// TIA Portal V17 export
// export: Created 2024-09-02T12:50:06.9482264Z, ExportSetting WithDefaults, DisplayName Totally Integrated Automation Portal, DisplayVersion V17, DisplayName TIA Portal Openness, DisplayVersion V17, DisplayName TIA Portal Version Control Interface, DisplayVersion V17, DisplayName STEP 7 Professional, DisplayVersion V17, DisplayName STEP 7 Safety, DisplayVersion V17, DisplayName WinCC Professional, DisplayVersion V17
FUNCTION "AnwFC1_FG01_Transport_OP70" : Void   // FC1281, LAD
TITLE = Transport
{ S7_Optimized_Access := 'TRUE' }
AUTHOR : VAF
FAMILY : SK
NAME : SK
VERSION : 0.1
// stored: AutoNumber false, IsIECCheckEnabled false, SetENOAutomatically false, UDAEnableTagReadback false
   VAR_TEMP
      Motion_Release : Bool;   // Motion permit
      Hand : Bool;
      Auto : Bool;
      t_ParityFault : Bool;
      t_ConfigFault : Bool;
      t_retval : Bool;
      "MM30/31_Home" : Bool;
      "MM30/31_Work" : Bool;
   END_VAR
BEGIN

REGION Network 1: Motion permit / Hand/ Auto
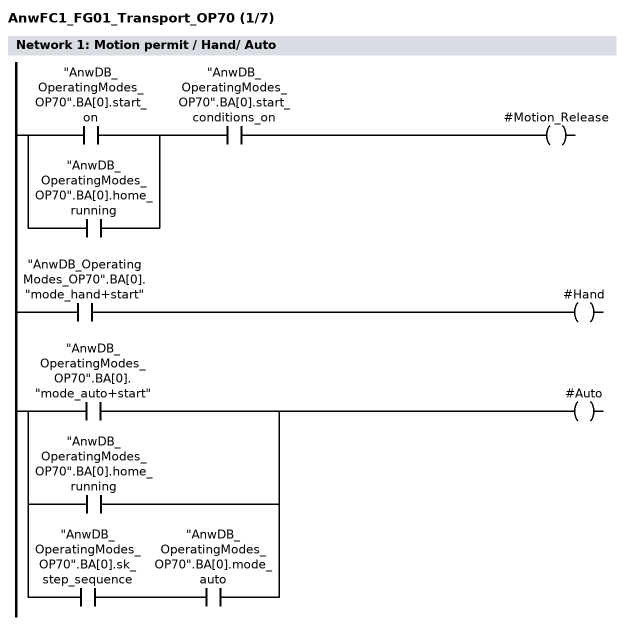
   RUNG wire#powerrail
      Contact( "AnwDB_OperatingModes_OP70".BA[0].start_on )
      wire#w1
      Contact( "AnwDB_OperatingModes_OP70".BA[0].start_conditions_on )
      Coil( #Motion_Release )
   END_RUNG
   RUNG wire#powerrail
      Contact( "AnwDB_OperatingModes_OP70".BA[0].home_running )
   END_RUNG wire#w1
   RUNG wire#powerrail
      Contact( "AnwDB_OperatingModes_OP70".BA[0]."mode_hand+start" )
      Coil( #Hand )
   END_RUNG
   RUNG wire#powerrail
      Contact( "AnwDB_OperatingModes_OP70".BA[0]."mode_auto+start" )
      wire#w2
      Coil( #Auto )
   END_RUNG
   RUNG wire#powerrail
      Contact( "AnwDB_OperatingModes_OP70".BA[0].home_running )
   END_RUNG wire#w2
   RUNG wire#powerrail
      Contact( "AnwDB_OperatingModes_OP70".BA[0].sk_step_sequence )
      Contact( "AnwDB_OperatingModes_OP70".BA[0].mode_auto )
   END_RUNG wire#w2
   // the same network as SCL:
   #Motion_Release := ("AnwDB_OperatingModes_OP70".BA[0].start_on OR "AnwDB_OperatingModes_OP70".BA[0].home_running) AND "AnwDB_OperatingModes_OP70".BA[0].start_conditions_on;
   #Hand := "AnwDB_OperatingModes_OP70".BA[0]."mode_hand+start";
   #Auto := "AnwDB_OperatingModes_OP70".BA[0]."mode_auto+start" OR "AnwDB_OperatingModes_OP70".BA[0].home_running OR ("AnwDB_OperatingModes_OP70".BA[0].sk_step_sequence AND "AnwDB_OperatingModes_OP70".BA[0].mode_auto);
END_REGION

REGION Network 2: Call of the step sequence
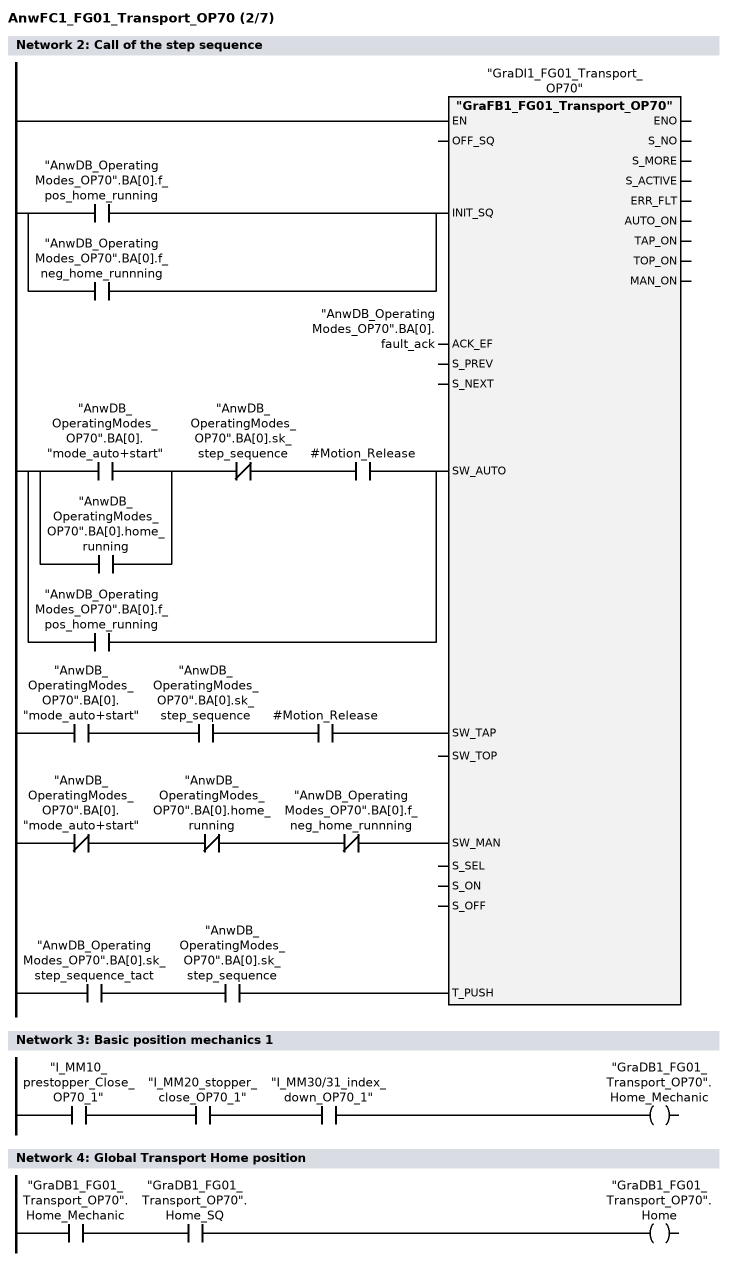
   RUNG wire#powerrail
      "GraDI1_FG01_Transport_OP70"(INIT_SQ := wire#w1, SW_AUTO := wire#w3, SW_TAP := wire#w4, SW_MAN := wire#w5, T_PUSH := wire#w6, OFF_SQ :=, ACK_EF := "AnwDB_OperatingModes_OP70".BA[0].fault_ack, S_PREV :=, S_NEXT :=, SW_TOP :=, S_SEL :=, S_ON :=, S_OFF :=, S_NO =>, S_MORE =>, S_ACTIVE =>, ERR_FLT =>, AUTO_ON =>, TAP_ON =>, TOP_ON =>, MAN_ON =>)
   END_RUNG
   RUNG wire#powerrail
      Contact( "AnwDB_OperatingModes_OP70".BA[0].f_pos_home_running )
   END_RUNG wire#w1
   RUNG wire#powerrail
      Contact( "AnwDB_OperatingModes_OP70".BA[0].f_neg_home_runnning )
   END_RUNG wire#w1
   RUNG wire#powerrail
      Contact( "AnwDB_OperatingModes_OP70".BA[0]."mode_auto+start" )
      wire#w2
      I_Contact( "AnwDB_OperatingModes_OP70".BA[0].sk_step_sequence )
      Contact( #Motion_Release )
   END_RUNG wire#w3
   RUNG wire#powerrail
      Contact( "AnwDB_OperatingModes_OP70".BA[0].home_running )
   END_RUNG wire#w2
   RUNG wire#powerrail
      Contact( "AnwDB_OperatingModes_OP70".BA[0].f_pos_home_running )
   END_RUNG wire#w3
   RUNG wire#powerrail
      Contact( "AnwDB_OperatingModes_OP70".BA[0]."mode_auto+start" )
      Contact( "AnwDB_OperatingModes_OP70".BA[0].sk_step_sequence )
      Contact( #Motion_Release )
   END_RUNG wire#w4
   RUNG wire#powerrail
      I_Contact( "AnwDB_OperatingModes_OP70".BA[0]."mode_auto+start" )
      I_Contact( "AnwDB_OperatingModes_OP70".BA[0].home_running )
      I_Contact( "AnwDB_OperatingModes_OP70".BA[0].f_neg_home_runnning )
   END_RUNG wire#w5
   RUNG wire#powerrail
      Contact( "AnwDB_OperatingModes_OP70".BA[0].sk_step_sequence_tact )
      Contact( "AnwDB_OperatingModes_OP70".BA[0].sk_step_sequence )
   END_RUNG wire#w6
   // the same network as SCL:
   "GraDI1_FG01_Transport_OP70"(INIT_SQ := "AnwDB_OperatingModes_OP70".BA[0].f_pos_home_running OR "AnwDB_OperatingModes_OP70".BA[0].f_neg_home_runnning,   // "GraFB1_FG01_Transport_OP70"
                           ACK_EF := "AnwDB_OperatingModes_OP70".BA[0].fault_ack,
                           SW_AUTO := (("AnwDB_OperatingModes_OP70".BA[0]."mode_auto+start" OR "AnwDB_OperatingModes_OP70".BA[0].home_running) AND NOT "AnwDB_OperatingModes_OP70".BA[0].sk_step_sequence AND #Motion_Release) OR "AnwDB_OperatingModes_OP70".BA[0].f_pos_home_running,
                           SW_TAP := "AnwDB_OperatingModes_OP70".BA[0]."mode_auto+start" AND "AnwDB_OperatingModes_OP70".BA[0].sk_step_sequence AND #Motion_Release,
                           SW_MAN := NOT "AnwDB_OperatingModes_OP70".BA[0]."mode_auto+start" AND NOT "AnwDB_OperatingModes_OP70".BA[0].home_running AND NOT "AnwDB_OperatingModes_OP70".BA[0].f_neg_home_runnning,
                           T_PUSH := "AnwDB_OperatingModes_OP70".BA[0].sk_step_sequence_tact AND "AnwDB_OperatingModes_OP70".BA[0].sk_step_sequence);
END_REGION

REGION Network 3: Basic position mechanics 1
   RUNG wire#powerrail
      Contact( "I_MM10_prestopper_Close_OP70_1" )
      Contact( "I_MM20_stopper_close_OP70_1" )
      Contact( "I_MM30/31_index_down_OP70_1" )
      Coil( "GraDB1_FG01_Transport_OP70".Home_Mechanic )
   END_RUNG
   // the same network as SCL:
   "GraDB1_FG01_Transport_OP70".Home_Mechanic := "I_MM10_prestopper_Close_OP70_1" AND "I_MM20_stopper_close_OP70_1" AND "I_MM30/31_index_down_OP70_1";
END_REGION

REGION Network 4: Global Transport Home position
   RUNG wire#powerrail
      Contact( "GraDB1_FG01_Transport_OP70".Home_Mechanic )
      Contact( "GraDB1_FG01_Transport_OP70".Home_SQ )
      Coil( "GraDB1_FG01_Transport_OP70".Home )
   END_RUNG
   // the same network as SCL:
   "GraDB1_FG01_Transport_OP70".Home := "GraDB1_FG01_Transport_OP70".Home_Mechanic AND "GraDB1_FG01_Transport_OP70".Home_SQ;
END_REGION

REGION Network 5: Finished message OK
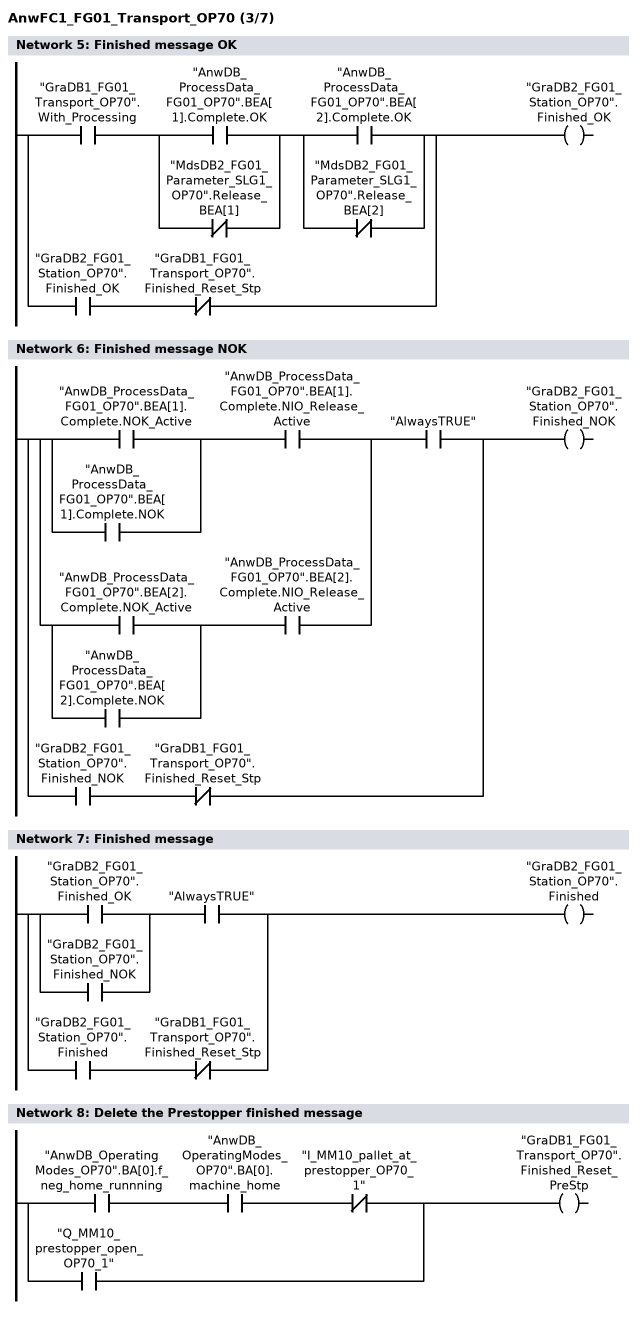
   RUNG wire#powerrail
      Contact( "GraDB1_FG01_Transport_OP70".With_Processing )
      wire#w1
      Contact( "AnwDB_ProcessData_FG01_OP70".BEA[1].Complete.OK )
      wire#w2
      Contact( "AnwDB_ProcessData_FG01_OP70".BEA[2].Complete.OK )
      wire#w3
      Coil( "GraDB2_FG01_Station_OP70".Finished_OK )
   END_RUNG
   RUNG wire#w1
      I_Contact( "MdsDB2_FG01_Parameter_SLG1_OP70".Release_BEA[1] )
   END_RUNG wire#w2
   RUNG wire#w2
      I_Contact( "MdsDB2_FG01_Parameter_SLG1_OP70".Release_BEA[2] )
   END_RUNG wire#w3
   RUNG wire#powerrail
      Contact( "GraDB2_FG01_Station_OP70".Finished_OK )
      I_Contact( "GraDB1_FG01_Transport_OP70".Finished_Reset_Stp )
   END_RUNG wire#w3
   // the same network as SCL:
   "GraDB2_FG01_Station_OP70".Finished_OK := ("GraDB1_FG01_Transport_OP70".With_Processing AND ("AnwDB_ProcessData_FG01_OP70".BEA[1].Complete.OK OR NOT "MdsDB2_FG01_Parameter_SLG1_OP70".Release_BEA[1]) AND ("AnwDB_ProcessData_FG01_OP70".BEA[2].Complete.OK OR NOT "MdsDB2_FG01_Parameter_SLG1_OP70".Release_BEA[2])) OR ("GraDB2_FG01_Station_OP70".Finished_OK AND NOT "GraDB1_FG01_Transport_OP70".Finished_Reset_Stp);
END_REGION

REGION Network 6: Finished message NOK
   RUNG wire#powerrail
      Contact( "AnwDB_ProcessData_FG01_OP70".BEA[1].Complete.NOK_Active )
      wire#w1
      Contact( "AnwDB_ProcessData_FG01_OP70".BEA[1].Complete.NIO_Release_Active )
      wire#w2
      Contact( "AlwaysTRUE" )
      wire#w4
      Coil( "GraDB2_FG01_Station_OP70".Finished_NOK )
   END_RUNG
   RUNG wire#powerrail
      Contact( "AnwDB_ProcessData_FG01_OP70".BEA[1].Complete.NOK )
   END_RUNG wire#w1
   RUNG wire#powerrail
      Contact( "AnwDB_ProcessData_FG01_OP70".BEA[2].Complete.NOK_Active )
      wire#w3
      Contact( "AnwDB_ProcessData_FG01_OP70".BEA[2].Complete.NIO_Release_Active )
   END_RUNG wire#w2
   RUNG wire#powerrail
      Contact( "AnwDB_ProcessData_FG01_OP70".BEA[2].Complete.NOK )
   END_RUNG wire#w3
   RUNG wire#powerrail
      Contact( "GraDB2_FG01_Station_OP70".Finished_NOK )
      I_Contact( "GraDB1_FG01_Transport_OP70".Finished_Reset_Stp )
   END_RUNG wire#w4
   // the same network as SCL:
   "GraDB2_FG01_Station_OP70".Finished_NOK := (((("AnwDB_ProcessData_FG01_OP70".BEA[1].Complete.NOK_Active OR "AnwDB_ProcessData_FG01_OP70".BEA[1].Complete.NOK) AND "AnwDB_ProcessData_FG01_OP70".BEA[1].Complete.NIO_Release_Active) OR (("AnwDB_ProcessData_FG01_OP70".BEA[2].Complete.NOK_Active OR "AnwDB_ProcessData_FG01_OP70".BEA[2].Complete.NOK) AND "AnwDB_ProcessData_FG01_OP70".BEA[2].Complete.NIO_Release_Active)) AND "AlwaysTRUE") OR ("GraDB2_FG01_Station_OP70".Finished_NOK AND NOT "GraDB1_FG01_Transport_OP70".Finished_Reset_Stp);
END_REGION

REGION Network 7: Finished message
   RUNG wire#powerrail
      Contact( "GraDB2_FG01_Station_OP70".Finished_OK )
      wire#w1
      Contact( "AlwaysTRUE" )
      wire#w2
      Coil( "GraDB2_FG01_Station_OP70".Finished )
   END_RUNG
   RUNG wire#powerrail
      Contact( "GraDB2_FG01_Station_OP70".Finished_NOK )
   END_RUNG wire#w1
   RUNG wire#powerrail
      Contact( "GraDB2_FG01_Station_OP70".Finished )
      I_Contact( "GraDB1_FG01_Transport_OP70".Finished_Reset_Stp )
   END_RUNG wire#w2
   // the same network as SCL:
   "GraDB2_FG01_Station_OP70".Finished := (("GraDB2_FG01_Station_OP70".Finished_OK OR "GraDB2_FG01_Station_OP70".Finished_NOK) AND "AlwaysTRUE") OR ("GraDB2_FG01_Station_OP70".Finished AND NOT "GraDB1_FG01_Transport_OP70".Finished_Reset_Stp);
END_REGION

REGION Network 8: Delete the Prestopper finished message
   RUNG wire#powerrail
      Contact( "AnwDB_OperatingModes_OP70".BA[0].f_neg_home_runnning )
      Contact( "AnwDB_OperatingModes_OP70".BA[0].machine_home )
      I_Contact( "I_MM10_pallet_at_prestopper_OP70_1" )
      wire#w1
      Coil( "GraDB1_FG01_Transport_OP70".Finished_Reset_PreStp )
   END_RUNG
   RUNG wire#powerrail
      Contact( "Q_MM10_prestopper_open_OP70_1" )
   END_RUNG wire#w1
   // the same network as SCL:
   "GraDB1_FG01_Transport_OP70".Finished_Reset_PreStp := ("AnwDB_OperatingModes_OP70".BA[0].f_neg_home_runnning AND "AnwDB_OperatingModes_OP70".BA[0].machine_home AND NOT "I_MM10_pallet_at_prestopper_OP70_1") OR "Q_MM10_prestopper_open_OP70_1";
END_REGION

REGION Network 9: Delete the stopper finished message
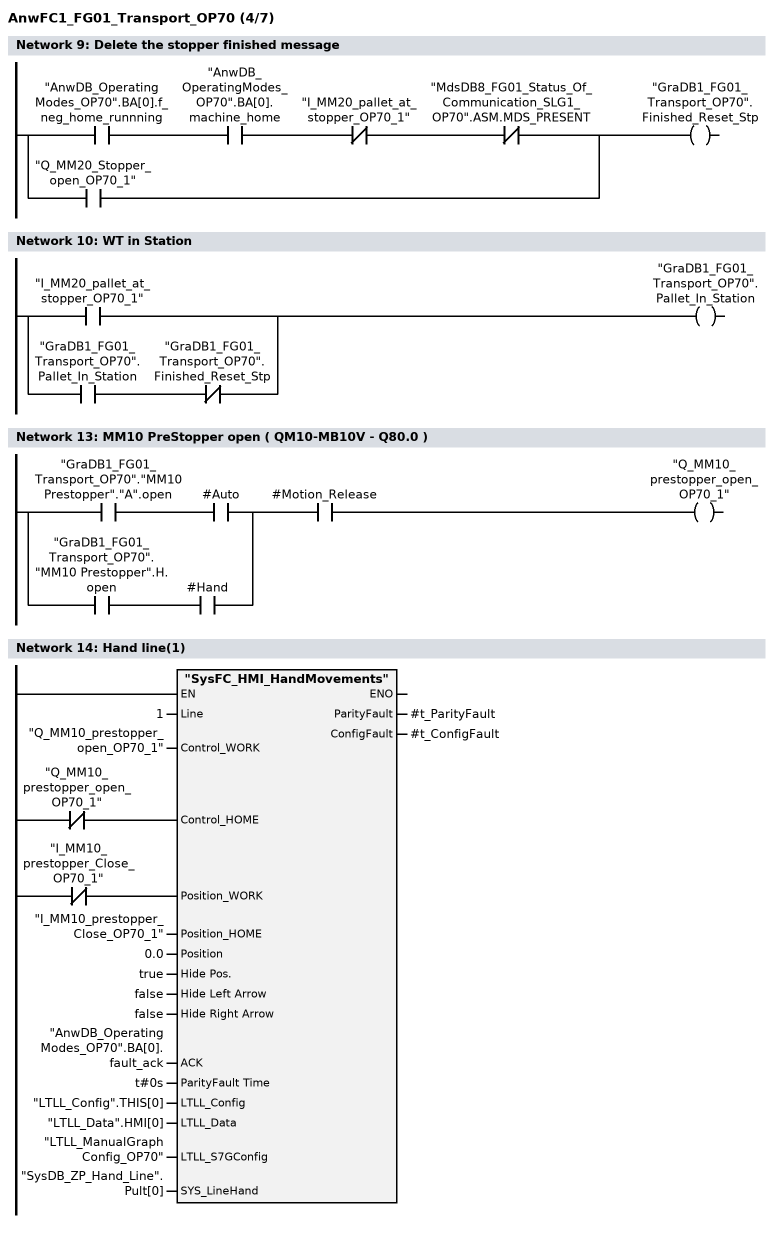
   RUNG wire#powerrail
      Contact( "AnwDB_OperatingModes_OP70".BA[0].f_neg_home_runnning )
      Contact( "AnwDB_OperatingModes_OP70".BA[0].machine_home )
      I_Contact( "I_MM20_pallet_at_stopper_OP70_1" )
      I_Contact( "MdsDB8_FG01_Status_Of_Communication_SLG1_OP70".ASM.MDS_PRESENT )
      wire#w1
      Coil( "GraDB1_FG01_Transport_OP70".Finished_Reset_Stp )
   END_RUNG
   RUNG wire#powerrail
      Contact( "Q_MM20_Stopper_open_OP70_1" )
   END_RUNG wire#w1
   // the same network as SCL:
   "GraDB1_FG01_Transport_OP70".Finished_Reset_Stp := ("AnwDB_OperatingModes_OP70".BA[0].f_neg_home_runnning AND "AnwDB_OperatingModes_OP70".BA[0].machine_home AND NOT "I_MM20_pallet_at_stopper_OP70_1" AND NOT "MdsDB8_FG01_Status_Of_Communication_SLG1_OP70".ASM.MDS_PRESENT) OR "Q_MM20_Stopper_open_OP70_1";
END_REGION

REGION Network 10: WT in Station
   RUNG wire#powerrail
      Contact( "I_MM20_pallet_at_stopper_OP70_1" )
      wire#w1
      Coil( "GraDB1_FG01_Transport_OP70".Pallet_In_Station )
   END_RUNG
   RUNG wire#powerrail
      Contact( "GraDB1_FG01_Transport_OP70".Pallet_In_Station )
      I_Contact( "GraDB1_FG01_Transport_OP70".Finished_Reset_Stp )
   END_RUNG wire#w1
   // the same network as SCL:
   "GraDB1_FG01_Transport_OP70".Pallet_In_Station := "I_MM20_pallet_at_stopper_OP70_1" OR ("GraDB1_FG01_Transport_OP70".Pallet_In_Station AND NOT "GraDB1_FG01_Transport_OP70".Finished_Reset_Stp);
END_REGION

REGION Network 11: ########### USER ###########
END_REGION

REGION Network 12: ########### SS_02_001_Setup ###########
END_REGION

REGION Network 13: MM10 PreStopper open ( QM10-MB10V - Q80.0 )
   RUNG wire#powerrail
      Contact( "GraDB1_FG01_Transport_OP70"."MM10 Prestopper"."A".open )
      Contact( #Auto )
      wire#w1
      Contact( #Motion_Release )
      Coil( "Q_MM10_prestopper_open_OP70_1" )
   END_RUNG
   RUNG wire#powerrail
      Contact( "GraDB1_FG01_Transport_OP70"."MM10 Prestopper".H.open )
      Contact( #Hand )
   END_RUNG wire#w1
   // the same network as SCL:
   "Q_MM10_prestopper_open_OP70_1" := (("GraDB1_FG01_Transport_OP70"."MM10 Prestopper"."A".open AND #Auto) OR ("GraDB1_FG01_Transport_OP70"."MM10 Prestopper".H.open AND #Hand)) AND #Motion_Release;
END_REGION

REGION Network 14: Hand line(1)
   RUNG wire#powerrail
      "SysFC_HMI_HandMovements"(Control_HOME := wire#w1, Position_WORK := wire#w2, Line := 1, Control_WORK := "Q_MM10_prestopper_open_OP70_1", Position_HOME := "I_MM10_prestopper_Close_OP70_1", Position := 0.0, "Hide Pos." := true, "Hide Left Arrow" := false, "Hide Right Arrow" := false, ACK := "AnwDB_OperatingModes_OP70".BA[0].fault_ack, "ParityFault Time" := t#0s, LTLL_Config := "LTLL_Config".THIS[0], LTLL_Data := "LTLL_Data".HMI[0], LTLL_S7GConfig := "LTLL_ManualGraphConfig_OP70", SYS_LineHand := "SysDB_ZP_Hand_Line".Pult[0], ParityFault => #t_ParityFault, ConfigFault => #t_ConfigFault)
   END_RUNG
   RUNG wire#powerrail
      I_Contact( "Q_MM10_prestopper_open_OP70_1" )
   END_RUNG wire#w1
   RUNG wire#powerrail
      I_Contact( "I_MM10_prestopper_Close_OP70_1" )
   END_RUNG wire#w2
   // the same network as SCL:
   "SysFC_HMI_HandMovements"(Line := 1,
                           Control_WORK := "Q_MM10_prestopper_open_OP70_1",
                           Control_HOME := NOT "Q_MM10_prestopper_open_OP70_1",
                           Position_WORK := NOT "I_MM10_prestopper_Close_OP70_1",
                           Position_HOME := "I_MM10_prestopper_Close_OP70_1",
                           Position := 0.0,
                           "Hide Pos." := true,
                           "Hide Left Arrow" := false,
                           "Hide Right Arrow" := false,
                           ACK := "AnwDB_OperatingModes_OP70".BA[0].fault_ack,
                           "ParityFault Time" := t#0s,
                           LTLL_Config := "LTLL_Config".THIS[0],
                           LTLL_Data := "LTLL_Data".HMI[0],
                           LTLL_S7GConfig := "LTLL_ManualGraphConfig_OP70",
                           SYS_LineHand := "SysDB_ZP_Hand_Line".Pult[0],
                           ParityFault => #t_ParityFault,
                           ConfigFault => #t_ConfigFault);
END_REGION

REGION Network 15: MM20 Stopper open ( QM20-MB20V - Q80.2 )
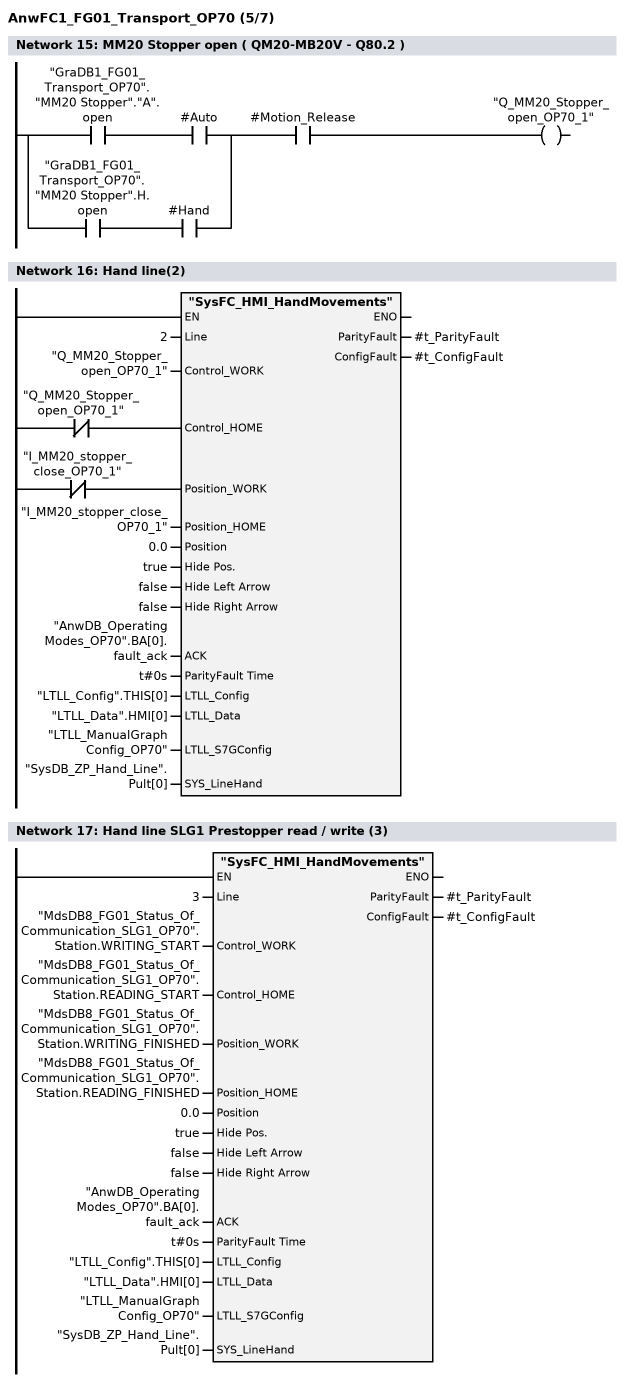
   RUNG wire#powerrail
      Contact( "GraDB1_FG01_Transport_OP70"."MM20 Stopper"."A".open )
      Contact( #Auto )
      wire#w1
      Contact( #Motion_Release )
      Coil( "Q_MM20_Stopper_open_OP70_1" )
   END_RUNG
   RUNG wire#powerrail
      Contact( "GraDB1_FG01_Transport_OP70"."MM20 Stopper".H.open )
      Contact( #Hand )
   END_RUNG wire#w1
   // the same network as SCL:
   "Q_MM20_Stopper_open_OP70_1" := (("GraDB1_FG01_Transport_OP70"."MM20 Stopper"."A".open AND #Auto) OR ("GraDB1_FG01_Transport_OP70"."MM20 Stopper".H.open AND #Hand)) AND #Motion_Release;
END_REGION

REGION Network 16: Hand line(2)
   RUNG wire#powerrail
      "SysFC_HMI_HandMovements"(Control_HOME := wire#w1, Position_WORK := wire#w2, Line := 2, Control_WORK := "Q_MM20_Stopper_open_OP70_1", Position_HOME := "I_MM20_stopper_close_OP70_1", Position := 0.0, "Hide Pos." := true, "Hide Left Arrow" := false, "Hide Right Arrow" := false, ACK := "AnwDB_OperatingModes_OP70".BA[0].fault_ack, "ParityFault Time" := t#0s, LTLL_Config := "LTLL_Config".THIS[0], LTLL_Data := "LTLL_Data".HMI[0], LTLL_S7GConfig := "LTLL_ManualGraphConfig_OP70", SYS_LineHand := "SysDB_ZP_Hand_Line".Pult[0], ParityFault => #t_ParityFault, ConfigFault => #t_ConfigFault)
   END_RUNG
   RUNG wire#powerrail
      I_Contact( "Q_MM20_Stopper_open_OP70_1" )
   END_RUNG wire#w1
   RUNG wire#powerrail
      I_Contact( "I_MM20_stopper_close_OP70_1" )
   END_RUNG wire#w2
   // the same network as SCL:
   "SysFC_HMI_HandMovements"(Line := 2,
                           Control_WORK := "Q_MM20_Stopper_open_OP70_1",
                           Control_HOME := NOT "Q_MM20_Stopper_open_OP70_1",
                           Position_WORK := NOT "I_MM20_stopper_close_OP70_1",
                           Position_HOME := "I_MM20_stopper_close_OP70_1",
                           Position := 0.0,
                           "Hide Pos." := true,
                           "Hide Left Arrow" := false,
                           "Hide Right Arrow" := false,
                           ACK := "AnwDB_OperatingModes_OP70".BA[0].fault_ack,
                           "ParityFault Time" := t#0s,
                           LTLL_Config := "LTLL_Config".THIS[0],
                           LTLL_Data := "LTLL_Data".HMI[0],
                           LTLL_S7GConfig := "LTLL_ManualGraphConfig_OP70",
                           SYS_LineHand := "SysDB_ZP_Hand_Line".Pult[0],
                           ParityFault => #t_ParityFault,
                           ConfigFault => #t_ConfigFault);
END_REGION

REGION Network 17: Hand line SLG1 Prestopper read / write (3)
   RUNG wire#powerrail
      "SysFC_HMI_HandMovements"(Line := 3, Control_WORK := "MdsDB8_FG01_Status_Of_Communication_SLG1_OP70".Station.WRITING_START, Control_HOME := "MdsDB8_FG01_Status_Of_Communication_SLG1_OP70".Station.READING_START, Position_WORK := "MdsDB8_FG01_Status_Of_Communication_SLG1_OP70".Station.WRITING_FINISHED, Position_HOME := "MdsDB8_FG01_Status_Of_Communication_SLG1_OP70".Station.READING_FINISHED, Position := 0.0, "Hide Pos." := true, "Hide Left Arrow" := false, "Hide Right Arrow" := false, ACK := "AnwDB_OperatingModes_OP70".BA[0].fault_ack, "ParityFault Time" := t#0s, LTLL_Config := "LTLL_Config".THIS[0], LTLL_Data := "LTLL_Data".HMI[0], LTLL_S7GConfig := "LTLL_ManualGraphConfig_OP70", SYS_LineHand := "SysDB_ZP_Hand_Line".Pult[0], ParityFault => #t_ParityFault, ConfigFault => #t_ConfigFault)
   END_RUNG
   // the same network as SCL:
   "SysFC_HMI_HandMovements"(Line := 3,
                           Control_WORK := "MdsDB8_FG01_Status_Of_Communication_SLG1_OP70".Station.WRITING_START,
                           Control_HOME := "MdsDB8_FG01_Status_Of_Communication_SLG1_OP70".Station.READING_START,
                           Position_WORK := "MdsDB8_FG01_Status_Of_Communication_SLG1_OP70".Station.WRITING_FINISHED,
                           Position_HOME := "MdsDB8_FG01_Status_Of_Communication_SLG1_OP70".Station.READING_FINISHED,
                           Position := 0.0,
                           "Hide Pos." := true,
                           "Hide Left Arrow" := false,
                           "Hide Right Arrow" := false,
                           ACK := "AnwDB_OperatingModes_OP70".BA[0].fault_ack,
                           "ParityFault Time" := t#0s,
                           LTLL_Config := "LTLL_Config".THIS[0],
                           LTLL_Data := "LTLL_Data".HMI[0],
                           LTLL_S7GConfig := "LTLL_ManualGraphConfig_OP70",
                           SYS_LineHand := "SysDB_ZP_Hand_Line".Pult[0],
                           ParityFault => #t_ParityFault,
                           ConfigFault => #t_ConfigFault);
END_REGION

REGION Network 18: MM30/31 Index unit up ( QM30-MB30V - Q81.0 )
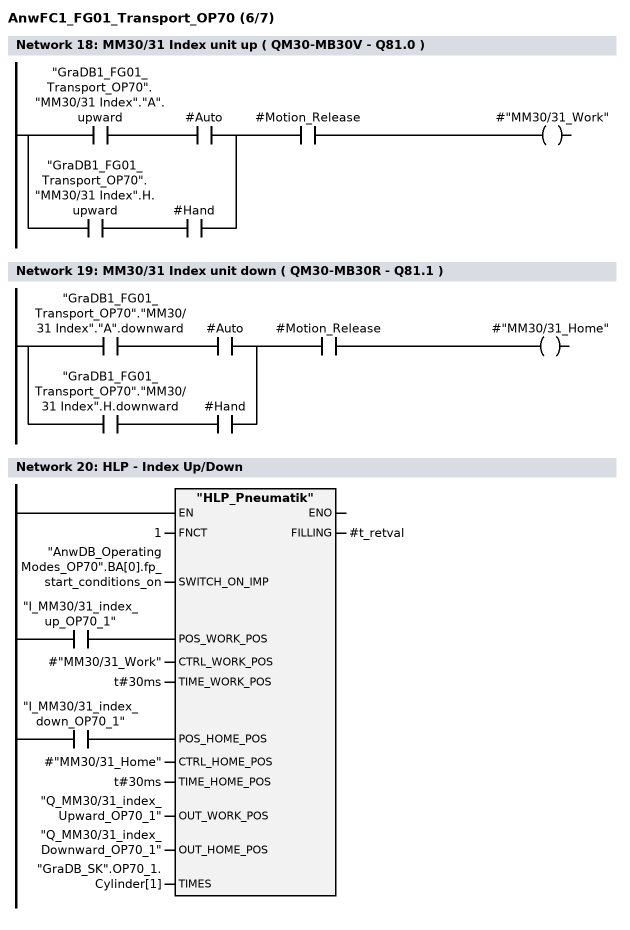
   RUNG wire#powerrail
      Contact( "GraDB1_FG01_Transport_OP70"."MM30/31 Index"."A".upward )
      Contact( #Auto )
      wire#w1
      Contact( #Motion_Release )
      Coil( #"MM30/31_Work" )
   END_RUNG
   RUNG wire#powerrail
      Contact( "GraDB1_FG01_Transport_OP70"."MM30/31 Index".H.upward )
      Contact( #Hand )
   END_RUNG wire#w1
   // the same network as SCL:
   #"MM30/31_Work" := (("GraDB1_FG01_Transport_OP70"."MM30/31 Index"."A".upward AND #Auto) OR ("GraDB1_FG01_Transport_OP70"."MM30/31 Index".H.upward AND #Hand)) AND #Motion_Release;
END_REGION

REGION Network 19: MM30/31 Index unit down ( QM30-MB30R - Q81.1 )
   RUNG wire#powerrail
      Contact( "GraDB1_FG01_Transport_OP70"."MM30/31 Index"."A".downward )
      Contact( #Auto )
      wire#w1
      Contact( #Motion_Release )
      Coil( #"MM30/31_Home" )
   END_RUNG
   RUNG wire#powerrail
      Contact( "GraDB1_FG01_Transport_OP70"."MM30/31 Index".H.downward )
      Contact( #Hand )
   END_RUNG wire#w1
   // the same network as SCL:
   #"MM30/31_Home" := (("GraDB1_FG01_Transport_OP70"."MM30/31 Index"."A".downward AND #Auto) OR ("GraDB1_FG01_Transport_OP70"."MM30/31 Index".H.downward AND #Hand)) AND #Motion_Release;
END_REGION

REGION Network 20: HLP - Index Up/Down
   RUNG wire#powerrail
      "HLP_Pneumatik"(POS_WORK_POS := wire#w1, POS_HOME_POS := wire#w2, FNCT := 1, SWITCH_ON_IMP := "AnwDB_OperatingModes_OP70".BA[0].fp_start_conditions_on, CTRL_WORK_POS := #"MM30/31_Work", TIME_WORK_POS := t#30ms, CTRL_HOME_POS := #"MM30/31_Home", TIME_HOME_POS := t#30ms, OUT_WORK_POS := "Q_MM30/31_index_Upward_OP70_1", OUT_HOME_POS := "Q_MM30/31_index_Downward_OP70_1", TIMES := "GraDB_SK".OP70_1.Cylinder[1], FILLING => #t_retval)
   END_RUNG
   RUNG wire#powerrail
      Contact( "I_MM30/31_index_up_OP70_1" )
   END_RUNG wire#w1
   RUNG wire#powerrail
      Contact( "I_MM30/31_index_down_OP70_1" )
   END_RUNG wire#w2
   // the same network as SCL:
   "HLP_Pneumatik"(FNCT := 1,
                   SWITCH_ON_IMP := "AnwDB_OperatingModes_OP70".BA[0].fp_start_conditions_on,
                   POS_WORK_POS := "I_MM30/31_index_up_OP70_1",
                   CTRL_WORK_POS := #"MM30/31_Work",
                   TIME_WORK_POS := t#30ms,
                   POS_HOME_POS := "I_MM30/31_index_down_OP70_1",
                   CTRL_HOME_POS := #"MM30/31_Home",
                   TIME_HOME_POS := t#30ms,
                   OUT_WORK_POS := "Q_MM30/31_index_Upward_OP70_1",
                   OUT_HOME_POS := "Q_MM30/31_index_Downward_OP70_1",
                   TIMES := "GraDB_SK".OP70_1.Cylinder[1],
                   FILLING => #t_retval);
END_REGION

REGION Network 21: Hand line(4)
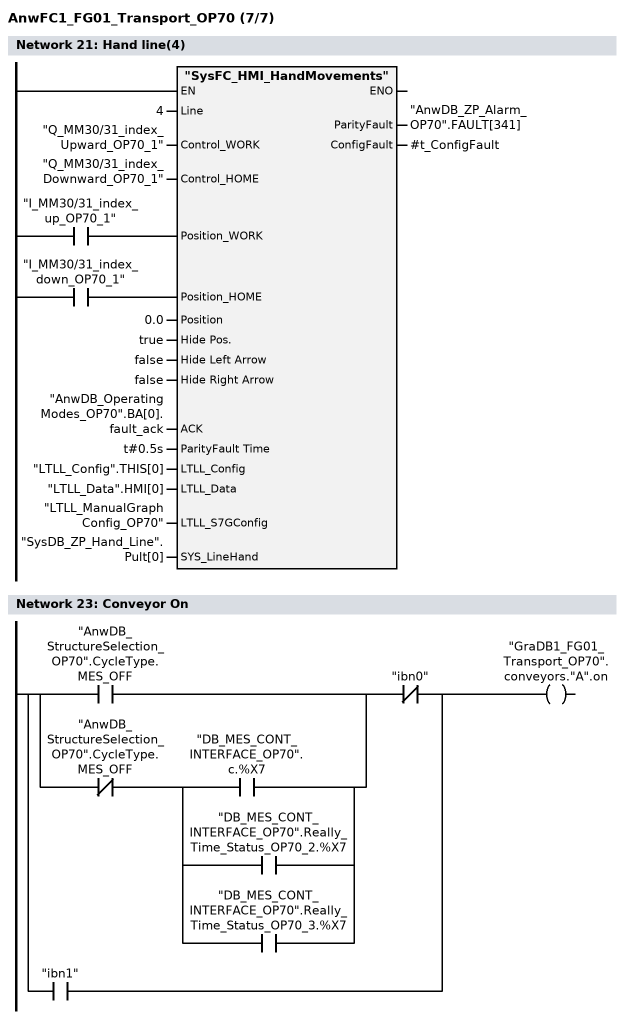
   RUNG wire#powerrail
      "SysFC_HMI_HandMovements"(Position_WORK := wire#w1, Position_HOME := wire#w2, Line := 4, Control_WORK := "Q_MM30/31_index_Upward_OP70_1", Control_HOME := "Q_MM30/31_index_Downward_OP70_1", Position := 0.0, "Hide Pos." := true, "Hide Left Arrow" := false, "Hide Right Arrow" := false, ACK := "AnwDB_OperatingModes_OP70".BA[0].fault_ack, "ParityFault Time" := t#0.5s, LTLL_Config := "LTLL_Config".THIS[0], LTLL_Data := "LTLL_Data".HMI[0], LTLL_S7GConfig := "LTLL_ManualGraphConfig_OP70", SYS_LineHand := "SysDB_ZP_Hand_Line".Pult[0], ParityFault => "AnwDB_ZP_Alarm_OP70".FAULT[341], ConfigFault => #t_ConfigFault)
   END_RUNG
   RUNG wire#powerrail
      Contact( "I_MM30/31_index_up_OP70_1" )
   END_RUNG wire#w1
   RUNG wire#powerrail
      Contact( "I_MM30/31_index_down_OP70_1" )
   END_RUNG wire#w2
   // the same network as SCL:
   "SysFC_HMI_HandMovements"(Line := 4,
                           Control_WORK := "Q_MM30/31_index_Upward_OP70_1",
                           Control_HOME := "Q_MM30/31_index_Downward_OP70_1",
                           Position_WORK := "I_MM30/31_index_up_OP70_1",
                           Position_HOME := "I_MM30/31_index_down_OP70_1",
                           Position := 0.0,
                           "Hide Pos." := true,
                           "Hide Left Arrow" := false,
                           "Hide Right Arrow" := false,
                           ACK := "AnwDB_OperatingModes_OP70".BA[0].fault_ack,
                           "ParityFault Time" := t#0.5s,
                           LTLL_Config := "LTLL_Config".THIS[0],
                           LTLL_Data := "LTLL_Data".HMI[0],
                           LTLL_S7GConfig := "LTLL_ManualGraphConfig_OP70",
                           SYS_LineHand := "SysDB_ZP_Hand_Line".Pult[0],
                           ParityFault => "AnwDB_ZP_Alarm_OP70".FAULT[341],
                           ConfigFault => #t_ConfigFault);
END_REGION

REGION Network 22: ##### Conveyors ON #####
END_REGION

REGION Network 23: Conveyor On
   RUNG wire#powerrail
      Contact( "AnwDB_StructureSelection_OP70".CycleType.MES_OFF )
      wire#w1
      I_Contact( "ibn0" )
      wire#w3
      Coil( "GraDB1_FG01_Transport_OP70".conveyors."A".on )
   END_RUNG
   RUNG wire#powerrail
      I_Contact( "AnwDB_StructureSelection_OP70".CycleType.MES_OFF )
      wire#w2
      Contact( "DB_MES_CONT_INTERFACE_OP70".c.%X7 )
   END_RUNG wire#w1
   RUNG wire#w2
      Contact( "DB_MES_CONT_INTERFACE_OP70".Really_Time_Status_OP70_2.%X7 )
   END_RUNG wire#w1
   RUNG wire#w2
      Contact( "DB_MES_CONT_INTERFACE_OP70".Really_Time_Status_OP70_3.%X7 )
   END_RUNG wire#w1
   RUNG wire#powerrail
      Contact( "ibn1" )
   END_RUNG wire#w3
   // the same network as SCL:
   "GraDB1_FG01_Transport_OP70".conveyors."A".on := (("AnwDB_StructureSelection_OP70".CycleType.MES_OFF OR (NOT "AnwDB_StructureSelection_OP70".CycleType.MES_OFF AND ("DB_MES_CONT_INTERFACE_OP70".c.%X7 OR "DB_MES_CONT_INTERFACE_OP70".Really_Time_Status_OP70_2.%X7 OR "DB_MES_CONT_INTERFACE_OP70".Really_Time_Status_OP70_3.%X7))) AND NOT "ibn0") OR "ibn1";
END_REGION
END_FUNCTION
